TYPE E_EndoscopeType :
(
	EndoscopeType_0:=1,
	EndoScopeType_30:=2
);
END_TYPE

(* stored: Version 1.1.0.1, ProductVersion 3.1.4024.12
   DUT E_EndoscopeType: Id {7bbe9ea4-82a3-4146-8613-f9d73d6783a3} *)
